ABB RobotStudio station: Estacion_herramienta.rsstn

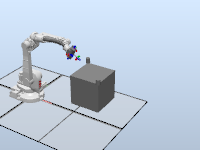
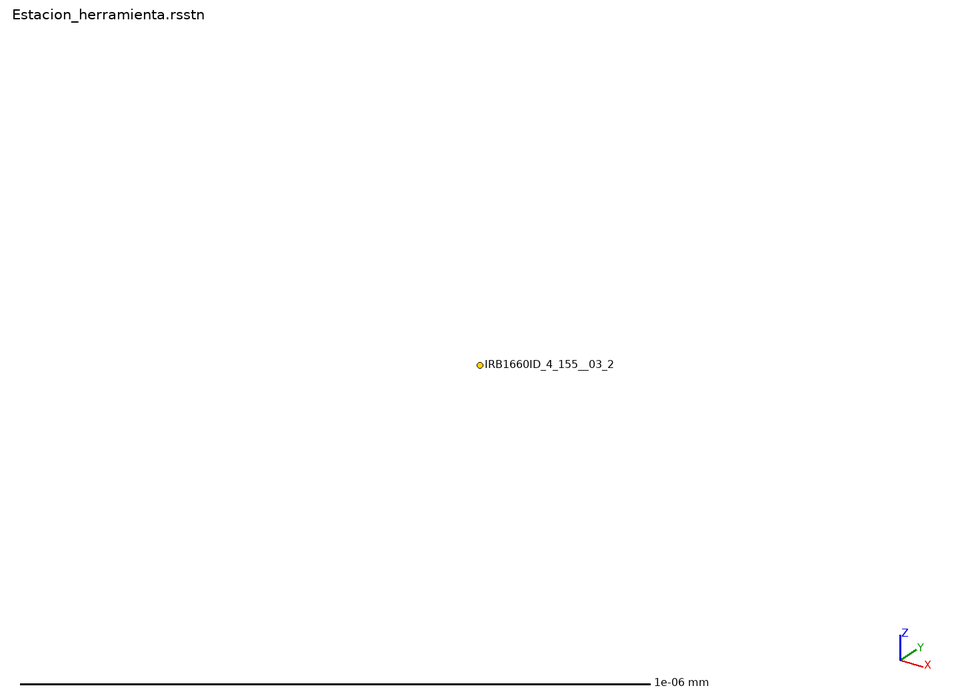
[picture v1: parts stored in the station drawn from their meshes, with robot base, taught points and paths (robot models come from the ABB library and are not in the file)]
Station Station (saved by RobotStudio 21.2.9526.0)
Controller Controlador8
  mechanical unit ROB_1: IRB1660ID_4_155__03_2, 6 joints, base frame (0, 0, 0) mm
Layout (positions relative to the parent item):
  - Cerrado1 [smart component, from Components\JointMover.rslib]
      properties: Mechanism=(none); Relative=false; Duration=1; J1=0.02; J2=0.02
  - Abierto1 [smart component, from Components\JointMover.rslib]
      properties: Mechanism=(none); Relative=false; Duration=1; J1=0; J2=0
  - IRB1660ID_4_155__03_2 [mechanism, from Robots\IRB1660ID_4_155__03.rslib] at (0, 0, 0) mm; joint values [0, 0, 0, 0, 0.5236, 0] (rad or m)
  - Efector_multiple [mechanism, from Libraries\Efector_multiple.rslib] at (944.87, 0, 1229) mm, rotated rx 180 ry 60 rz 180 deg
  - Pieza_17 [part] at (300, 300, 600) mm, size 80 x 79.4 x 100 mm
  - Cilindros [part] at (900, -300, 600) mm, size 80 x 79.4 x 100 mm
  - Pieza_18 [part], size 600 x 600 x 600 mm
Attachment: Efector_multiple is attached to IRB1660ID_4_155__03_2 / Link6
Station signals: DI Abrir_P1, DI Cerrar_P1, DI Abrir_P2, DI Cerrar_P2
Station logic (signal -> signal, property => property):
  Station.Abrir_P1 -> Abierto1.Execute
  Station.Cerrar_P1 -> Cerrado1.Execute
Targets, tools, work objects and paths stored in the station, written as RAPID:
! task T_ROB1
MODULE CalibData
  PERS tooldata Pinza_1:=[TRUE,[[-100,0,70],[0.707106781,0,-0.707106781,0]],[1,[0,0,1],[1,0,0,0],0,0,0]];
  PERS tooldata Pinza_2:=[TRUE,[[100,0,70],[0.707106781,0,0.707106781,0]],[1,[0,0,1],[1,0,0,0],0,0,0]];
  PERS tooldata Punta_rev:=[TRUE,[[0,0,200],[1,0,0,0]],[1,[0,0,1],[1,0,0,0],0,0,0]];
  PERS tooldata Limpiador:=[TRUE,[[0,-50,70],[1,0,0,0]],[1,[0,0,1],[1,0,0,0],0,0,0]];
ENDMODULE

